// TIA Portal V17 export
// export: Created 2026-04-13T11:12:42.142207Z, ExportSetting WithDefaults, DisplayName Totally Integrated Automation Portal, DisplayVersion V17 Update 4, DisplayName TIA Portal Openness, DisplayVersion V17 Update 4, DisplayName TIA Portal Version Control Interface, DisplayVersion V17, DisplayName SINAMICS Startdrive Advanced, DisplayVersion V17, DisplayName SINAMICS Startdrive G130, G150, S120, S150, SINAMICS MV, S210, DisplayVersion V17, DisplayName SINAMICS Startdrive G110M, G120, G120C, G120D, G120P, G115D, DisplayVersion V17, DisplayName STEP 7 Professional, DisplayVersion V17 Update 4, DisplayName STEP 7 Safety, DisplayVersion V17, DisplayName WinCC Professional, DisplayVersion V17 Update 4
FUNCTION_BLOCK "时间累计"   // FB66, SCL
{ S7_Optimized_Access := 'TRUE' }
VERSION : 0.1
// stored: AutoNumber true, IsIECCheckEnabled false, IsRetainMemResEnabled false, MemoryReserve 100, SetENOAutomatically false, UDAEnableTagReadback false
   VAR_INPUT
      start : Bool;
      reset : Bool;
   END_VAR
   VAR_OUTPUT
      h : Int;
      "m" : Int;
      s : Int;
   END_VAR
   VAR
      T1S : TON_TIME;
   END_VAR
BEGIN

   IF #start AND #T1S.Q THEN
       #s := #s + 1;
   END_IF;
   IF #reset THEN
       #h := 0;
       #m := 0;
       #s := 0;
   END_IF;
   IF #s >= 60 THEN
       #m := #m + 1;
       #s := 0;
   END_IF;

   IF #m >= 60 THEN
       #h := #h + 1;
       #m := 0;
   END_IF;

   #T1S(IN := NOT #T1S.Q,
        PT := T#1S);
END_FUNCTION_BLOCK
